(* IEC 61131-3 sources: SigmatekTestframework/src/Class/CXmlTestReport, 1 file *)

(* ---- CXmlTestReport.st ---- *)
#define XML_VERSION     "<?xml version=$221.0$22 encoding=$22UTF-8$22?>"

(*!
<Class
	Name               = "CXmlTestReport"
	Revision           = "1.0"
	RealtimeTask       = "false"
	CyclicTask         = "false"
	BackgroundTask     = "false"
	Sigmatek           = "false"
	OSInterface        = "false"
	HighPriority       = "false"
	Automatic          = "false"
	UpdateMode         = "Prescan"
	SharedCommandTable = "true"
	Objectsize         = "(510,120)">
	<Channels>
		<Client Name="ViewDetails" Required="false" Internal="false" Comment="0 = short report&#13;&#10;1 = extended report"/>
	</Channels>
	<Network Name="CXmlTestReport">
		<!-- List of Components in this network -->
		<Components>
			<Object
				Name       = "_base"
				Class      = "CTestReportBase"
				Position   = "(218,120)"
				Visualized = "false">
				<Channels>
					<Server Name="Registered"/>
					<Client Name="clib"/>
					<Client Name="File"/>
					<Client Name="System"/>
				</Channels>
			</Object>
		</Components>
		<Comments>
		</Comments>
		<!-- List of Connections in this network -->
		<Connections>
			<Connection Source="this.Registered" Destination="_base.Registered" Vertices="(690,210),(518,210),"/>
			<Connection Source="_base.File" Destination="this.File" Vertices="(218,210),(38,210),"/>
		</Connections>
		<!-- Headerfiles -->
		<Options>
		</Options>
	</Network>
</Class>
*)
#pragma using CTestReportBase

CXmlTestReport : CLASS
: CTestReportBase
  //Servers:
  //Clients:
	ViewDetails 	: CltCh_DINT;
  //Variables:
  //Functions:

	FUNCTION VIRTUAL BuildFile
		VAR_OUTPUT
			eRetcode 	: ERetCode_t;
		END_VAR;

	FUNCTION VIRTUAL getFileName
		VAR_INPUT
			pFileName 	: ^CHAR;
			pFilePath 	: ^CHAR;
		END_VAR
		VAR_OUTPUT
			eRetcode 	: ERetCode_t;
		END_VAR;
  //Tables:
	FUNCTION @STD
		VAR_OUTPUT
			ret_code	: CONFSTATES;
		END_VAR;
	FUNCTION GLOBAL TAB @CT_;
END_CLASS;

//Exclude-SccX
(*
 **********************************************************************
 * \file CXmlTestReport.st
 *
 * Creates a simple XML-File as report
 *
 * Copyright (c) 2016,Hoox.Software, Helmbrechts
 * All Rights Reserved.
 *
 * Created on: 01.06.2016
 *     Author: dressel
 *
 **********************************************************************
 *)

//*********************************************************************
//
//
//
//
//*********************************************************************
FUNCTION VIRTUAL CXmlTestReport::getFileName
	VAR_INPUT
		pFileName 	: ^CHAR;
		pFilePath 	: ^CHAR;
	END_VAR
	VAR_OUTPUT
		eRetcode 	: ERetCode_t;
	END_VAR

   _strcpy(dest:= pFilePath, src:= "C:\Testrun");
   _strcpy(dest:= pFileName, src:= "Testlog1.xml");

   eRetcode := eDone;

END_FUNCTION

//*********************************************************************
//
//
//
//
//*********************************************************************
FUNCTION VIRTUAL CXmlTestReport::BuildFile
	VAR_OUTPUT
		eRetcode 	: ERetCode_t;
	END_VAR
   VAR
   	u32Suites : UDINT;
   END_VAR

   clearBuffer();

   addString(XML_VERSION);
   writeBuffer();

   // <Created Date=dd.mm.yy Time=hh.mm.ss>
   addString("</Created Date=");
   addDate(#m_sSysDate);
   addString(" Time=");
   addTime(#m_sSysTime);
   addString(" >");
   writeBuffer();

   addString("<TestReport NbSuites=");
   addValue(m_pTestLib^.NbSuites$DINT);
   addString(" NbTests=");
   addValue(m_pTestLib^.NbRun$DINT);
   addString(" NbPassed=");
   addValue(m_pTestLib^.NbPassed$DINT);
   addString(" NbFailed=");
   addValue(m_pTestLib^.NbFailed$DINT);
   addString(" >");

   writeBuffer();

   if ViewDetails = 1 then

      u32Suites := m_pTestLib^.NbSuites;

      while u32Suites > 0 do

         addString("$09<Testsuite>");
         writeBuffer();

         addString("$09</Testsuite>");
         writeBuffer();

         u32Suites -= 1;

      end_while;

   end_if;

   addString("</TestReport>");
   writeBuffer();

   eRetcode := eDone;

END_FUNCTION
